FUNCTION_BLOCK FB_Abfuellmodul
VAR_INPUT
    bEnable  : BOOL;
    bExecute : BOOL;
    bReset   : BOOL;
    // Status-Rückmeldungen der Abteilungsleiter
	
    // bVereinzelungDone : BOOL;
    // bTransportDone    : BOOL;
    // bDisp1Done        : BOOL;
    // bDisp2Done        : BOOL;
    // bDisp3Done        : BOOL;
	
	// Error handling
	//bTransportError : BOOL; 
    
END_VAR
VAR_OUTPUT
    eState   : E_State;
    
    
END_VAR
VAR
    nState : INT;
    i      : INT; // Unser Stations-Zähler (1, 2, 3)
	bFlascheAktiv : BOOL;	// Flasche im System?
	
	fbVereinzelung : FB_Vereinzelung; 
    fbTransport    : FB_Transport;
    fbDisp1        : FB_Dispenser;
    fbDisp2        : FB_Dispenser;
    fbDisp3        : FB_Dispenser;
	
	// Start-Befehle
    bStartVereinzelung : BOOL;
    bStartTransport    : BOOL;
    nZielStation       : INT;     // Welcher Extruder ist das Ziel?
    bStartDisp1        : BOOL;
    bStartDisp2        : BOOL;
    bStartDisp3        : BOOL;
	
	bStop : Bool;
	nMemState: INT;
END_VAR

IF NOT bEnable THEN
    nState := 0;
	eState := E_State.Off;
ELSIF fbTransport.bError AND nState <> 99 THEN
	nMemState := nState;
    nState := 99;
END_IF

// neu 
IF bStop THEN
	nMemState := nState;
END_IF

CASE nState OF
    0: // Start / Bereit
        IF bEnable THEN
            eState := E_State.Ready;
        END_IF
		
        bStartVereinzelung := FALSE;
        bStartTransport    := FALSE;
        bStartDisp1        := FALSE;
        bStartDisp2        := FALSE;
        bStartDisp3        := FALSE;

        IF bExecute THEN
            nState := 10;
        END_IF

    10: // "Vereinzeln der Flasche"
        eState := E_State.Production;
        // --- 1. INTELLIGENTE SUCHE: Steht die Flasche exakt am Sensor? ---
        IF IFC_HW.bBandSens1 THEN
            i := 1; nState := 30; 
        ELSIF IFC_HW.bBandSens2 THEN
            i := 2; nState := 30; 
        ELSIF IFC_HW.bBandSens3 THEN
            i := 3; nState := 30; 
        ELSIF IFC_HW.bBandSens4 THEN
            nState := 40; 

        // --- 2. Suche im Gedächtnis (Der Blinde Fleck) ---
        ELSIF bFlascheAktiv THEN
            // Sensoren sehen nichts, aber da ist eine Flasche!
            // WICHTIG: Wohin war sie gerade unterwegs?
            IF i < 4 THEN
                nState := 20; // Sie war auf dem Weg zu einem Extruder (1, 2 oder 3)
            ELSE
                nState := 40; // Sie war schon auf der Zielgeraden zum Roboter (Station 4)
            END_IF
			
        // --- 3. NORMALBETRIEB: Keine alte Flasche im System ---
        ELSE
            bStartVereinzelung := TRUE;
        END_IF

        IF fbVereinzelung.eStateOut = E_State.Done THEN
            bFlascheAktiv := TRUE;
            i := 1;                      // Zähler auf ersten Extruder setzen!
            nState := 20;
        END_IF

    20: // "Fördern zu Extruder i"
		eState := E_State.Production;
        nZielStation := i; // Dem Transport das Ziel (1, 2 oder 3) mitteilen
        bStartTransport := TRUE;

        IF fbTransport.eState = E_State.Done THEN
            
           	IF i = 1 THEN
                bStartVereinzelung := FALSE; // Vereinzelung darf nächste Flasche holen
            END_IF
            
            bStartTransport := FALSE;
            nState := 30;
        END_IF

    30: // "Extruder i Start"
		eState := E_State.Production;
        // Welcher Dispenser muss gestartet werden?
        IF i = 1 THEN bStartDisp1 := TRUE; END_IF
        IF i = 2 THEN bStartDisp2 := TRUE; END_IF
        IF i = 3 THEN bStartDisp3 := TRUE; END_IF

        // Warten, bis der jeweilige Extruder "fertig" meldet
        IF (i = 1 AND fbDisp1.eState = E_State.Done) OR
           (i = 2 AND fbDisp2.eState = E_State.Done) OR
           (i = 3 AND fbDisp3.eState = E_State.Done) THEN
            
            // Befehle wieder wegnehmen
            bStartDisp1 := FALSE;
            bStartDisp2 := FALSE;
            bStartDisp3 := FALSE;

            // Zähler erhöhen! (i = i + 1)
            i := i + 1;

            // Prüfen, ob wir alle 3 Extruder durch haben
            IF i < 4 THEN
                nState := 20; // Zurück zu Schritt 20: Fördern zum NÄCHSTEN Extruder!
            ELSE
                nState := 40; // Alle 3 Farben sind drin! Weiter zur Übergabe.
            END_IF
        END_IF

    40: // "Übergabe zu Portalroboter" / Station 4 (PDF S.3)
		eState := E_State.Production;
        nZielStation := 4;
        bStartTransport := TRUE;

        IF fbTransport.eState = E_State.Done THEN
            bStartTransport := FALSE;
            nState := 50;
        END_IF

    50: // Done
        eState := E_State.Done;
		
		bFlascheAktiv := FALSE;

        IF NOT bExecute THEN
            nState := 0; // Warten auf die nächste Flasche
        END_IF
	
	99: // Error
        eState := E_State.Error; 
        IF NOT fbTransport.bError THEN
            nState := nMemState; // Nach Reset zurück zum alten zustand
        END_IF
        
END_CASE



// FBs

fbVereinzelung(
    bEnable  := bEnable,
    bExecute := bStartVereinzelung, // Interne Variable
    bSens1   := IFC_HW.bEinzelSens1,
    bSens2   := IFC_HW.bEinzelSens2,
    bSens3   := IFC_HW.bEinzelSens3
);

fbTransport(
    bEnable  := bEnable,
    bExecute := bStartTransport,    // Interne Variable
    bReset   := bReset,
    nStation := nZielStation,       // Interne Variable
    bSens1   := IFC_HW.bBandSens1,
    bSens2   := IFC_HW.bBandSens2,
    bSens3   := IFC_HW.bBandSens3,
    bSens4   := IFC_HW.bBandSens4
);

// Direktes Beschreiben der Hardware-Ausgänge für den Transport
IFC_HW.bBandHub1 := fbTransport.bHub1;
IFC_HW.bBandHub2 := fbTransport.bHub2;
IFC_HW.bBandHub3 := fbTransport.bHub3;

fbDisp1(
    ax := IFC_HW.ax_Extruder1,
    bEnable := bEnable,
    bExecute := bStartDisp1,        // Interne Variable
    bSensFlasche := IFC_HW.bBandSens1,
    iFuellstand := IFC_HW.iFillSens1,
    iLimit := 80
);

fbDisp2(
    ax := IFC_HW.ax_Extruder2,
    bEnable := bEnable,
    bExecute := bStartDisp2,        // Interne Variable
    bSensFlasche := IFC_HW.bBandSens2,
    iFuellstand := IFC_HW.iFillSens2,
    iLimit := 80
);

fbDisp3(
    ax := IFC_HW.ax_Extruder3,
    bEnable := bEnable,
    bExecute := bStartDisp3,        // Interne Variable
    bSensFlasche := IFC_HW.bBandSens3,
    iFuellstand := IFC_HW.iFillSens3,
    iLimit := 80
);

END_FUNCTION_BLOCK

(* stored: Version 1.1.0.1
   POU FB_Abfuellmodul: Id {c9826859-957f-4a6e-8c24-b0c6a8923961}, SpecialFunc None *)
